(* CoDeSys 2.3.9.37 project: Cap11_5.pro *)
(* Libraries: Standard.lib 4.10.05 12:14:46, IecSfc.lib 13.4.06 16:51:28 *)

(* POU PLC_PRG, SFC *)
PROGRAM PLC_PRG
VAR
       (* Entradas *)
	A: BOOL;
	B: BOOL;
      (* Salidas *)
	Salida: BOOL;
      (* Otras *)
	MiTempo: TON;
	TiempoActual: TIME;
END_VAR
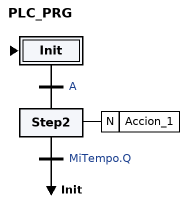
INITIAL_STEP Init:
END_STEP
TRANSITION FROM Init TO Step2 := A;
END_TRANSITION
STEP Step2:
	Accion_1(N);
END_STEP
TRANSITION FROM Step2 TO Init := MiTempo.Q;
END_TRANSITION
END_PROGRAM
ACTION Accion_1:
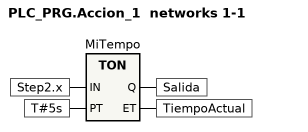
_FBD_ (* Function Block Diagram *)
NETWORK 1
	MiTempo:TON(IN: Step2.x, PT: T#5s, ET => TiempoActual) => Salida
_END_FBD_
(* the same logic as Structured Text *)
(* Network 1 *)
MiTempo(IN := Step2.x, PT := T#5s);
TiempoActual := MiTempo.ET;
Salida := MiTempo.Q;
END_ACTION

(* Visualisation Visu
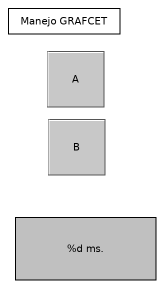
button at (131,60)-(188,116): text "A"; taps PLC_PRG.A
button at (132,128)-(189,184): text "B"; taps PLC_PRG.B
rectangle at (92,17)-(204,43): text "Manejo GRAFCET"
rounded rectangle at (99,226)-(240,289): text "%d ms."; shows PLC_PRG.MiTempo.ET; alarm colour if PLC_PRG.Salida
*)
